Fanuc KAREL source: kb00186.KL

-- PROVISIONAL review KL for V770-1; original PC SHA256 f5bdb837b3ffdb7368ff3f2b13d2f538613cd3450aa22bb94f4485909b3e0fda
-- Incomplete behavior may be omitted. Consult companion uncertainty JSON. Do not deploy.
PROGRAM KB00186
%NOLOCKGROUP
VAR
  P1 : REAL
  RESULT : REAL
BEGIN
  -- UNRESOLVED_PC offsets 5-16; opcodes 2E,23
  -- UNRESOLVED_PC offsets 21-36; opcodes 27,22,76,23
  -- UNRESOLVED_PC offsets 41-45; opcodes 7F
END KB00186
